INTERFACE SpindleControl

METHOD Run : BOOL
END_METHOD

METHOD SetSpeed : BOOL
VAR_INPUT
	Speed : UINT;
END_VAR
END_METHOD

METHOD Stop : BOOL
END_METHOD

END_INTERFACE

(* stored: Version 1.1.0.1, ProductVersion 3.1.4022.16
   Itf SpindleControl: Id {df9af8cd-f926-49bc-9ede-9a0faf189bc9}
   Method Run: Id {bde1c9a9-ee7f-4e70-897d-f6e0e05beb6a}
   Method SetSpeed: Id {cb2af7f9-4e6c-4e88-9d58-7c04bcf58105}
   Method Stop: Id {775584b9-1b67-4b01-a066-f4712b5973a1} *)
